# EPICS autosave request: opticsApp/Db/flexCapSensor_settings.req
$(P)$(C):posCalc.PREC
$(P)$(C):pos.PREC
$(P)$(C):umPerV.VAL
$(P)$(C):umPerV.PREC
$(P)$(C):offset.VAL
$(P)$(C):offset.PREC
